INTERFACE I_LensCompounder EXTENDS I_Fallible


METHOD Compound
VAR_INPUT
    FocalLength : I_QuantityLREAL;
    Multiplier : INT;
END_VAR
VAR_IN_OUT
    FocalLengthCompounded : FB_QuantityLREALPublic(Units := 'm');
END_VAR
END_METHOD


METHOD Reset
END_METHOD

END_INTERFACE

(* stored: Version 1.1.0.1
   Itf I_LensCompounder: Id {189c73c1-218b-43e0-9071-b2f04c9c5f2f}
   Method Compound: Id {d26e5efe-a98a-494e-9f0a-b13836021aba}
   Method Reset: Id {60082cfe-04c6-4032-849f-43568023ac1a} *)
